Fanuc KAREL source: kt00273.KL

-- PROVISIONAL review KL for V770-1; original PC SHA256 ce0a61d13d9ba93acf2b9a241810c0506cb13ac559e03b18a05d0b92f28b3b2d
-- Incomplete behavior may be omitted. Consult companion uncertainty JSON. Do not deploy.
PROGRAM KT00273
%NOLOCKGROUP
VAR
  OUT : BOOLEAN
-- UNRESOLVED_DECL H1 type=002017
-- UNRESOLVED_DECL Y2 type=002018
BEGIN
  -- UNRESOLVED_PC offsets 5-19; opcodes 2E,22,9D,33,B4
  -- UNRESOLVED_PC offsets 24-38; opcodes 2E,22,9D,33,B2
  -- UNRESOLVED_PC offsets 43-68; opcodes 22,9D,33,B3,22,9D,33,B1,57,23
  -- UNRESOLVED_PC offsets 73-77; opcodes 7F
END KT00273
